{attribute addProperty BoxType "EP1122-0001-0016"}
{attribute addProperty Id "A_0025_EP1122_0001_0017A_0025_EP1122_0001_0017_6C56F6A91080068719478086"}
{attribute addProperty CRC "96324977"}
{attribute addProperty SizeInBites "10800"}
{attribute addProperty SizeInBytes "68719478086"}
TYPE A_0024_EP1122_0001_0016_05BDCD71 EXTENDS EP1122_179A0949 :
STRUCT
	{attribute addProperty Name "A_0025_EP1122_0001_0017"}
	A_0025_EP1122_0001_0017 : A_0025_EP1122_0001_0017_6C56F6A9;
END_STRUCT
END_TYPE

(* stored: Version 1.2.0.0, ProductVersion 3.1.4024.9
   DUT A_0024_EP1122_0001_0016_05BDCD71: Id {f7e19aa5-70d7-46c5-892c-2aaec7a36c13} *)
